TYPE ST_GHMI :
STRUCT
  bStartButton      		  : BOOL;
  bStopButton       		  : BOOL;
  bResetButton      		  : BOOL;
  bAbortButton      		  : BOOL;
  bClearButton      		  : BOOL;
  nIndexFrame       		  : INT := 0;
  nIndexFrameAdmin        : INT := 0;
  nIndexFrameHome   		  : INT := 0;
  bPopUpModulPresent		  : BOOL;
  bPopUpHoming      		  : BOOL;
  bPopUpExtractorAborted  : BOOL;
	bPopUpInsertModulesLine	: BOOL;
  bRestart          		  : BOOL;
  bShutdown          		  : BOOL;
	sBtnAdmin								: STRING(32);
END_STRUCT
END_TYPE

(* stored: Version 1.1.0.1, ProductVersion 3.1.4024.12
   DUT ST_GHMI: Id {6205cda5-0483-481f-8601-06879509a1f4} *)
